Staubli VAL3: cycle_stop.pgx

program cycle_stop()
begin
  logMsg("[KERNEL] PLC:Stop Cycle")
  if cycleStatus:bCycle or cycleStatus:bSimulation
    // stop bit
    cycleStatus:bToStop=true
    watch(cycleStatus:bToStop==false,1)
  endIf
end
